PROGRAM MAIN
VAR
	
	fMotorRunningStatus : BOOL;
	fbFixedMotor1 : FB_FixedMotor;
	iMotor : I_Motor;
	fbVariableMotor1 : FB_VariableMotor;
	
	fbVariableMotor2 : FB_VariableSpeedMotor;
	bRun : BOOL := TRUE;
	
	fbLight1 : FB_Light;
	
	fSpeed : REAL := 34.343;
	bType : BOOL;
END_VAR


MotorController(fbFixedMotor1, bRun,fSpeed );
MotorController (fbVariableMotor1, bRun, fSpeed);
MotorController (fbVariableMotor2 , bRun , fSpeed);
fbVariableMotor2.M_SetSpeed(fspeed);
bType := __QUERYINTERFACE(fbVariableMotor2 , iMotor);

END_PROGRAM

(* stored: Version 1.1.0.1, ProductVersion 3.1.4024.16
   POU MAIN: Id {d8671499-345b-4312-95fc-c382a6413344}, SpecialFunc None *)
